//==================================================================================================
//							Beckhoff Automation Poland
//									3.01.2022
//	Function block running PLC CAM procedure using hardware limit switch
//	Library: Tc3_MC2_AdvancedHoming, Tc2_MC2, 
//
//  v1.0	|| TC v 3.1.4024.22		|| First edition 
//==================================================================================================
FUNCTION_BLOCK FB_HomingLimitSwitch
VAR_IN_OUT
	Axis 										: Tc2_MC2.AXIS_REF;
END_VAR
VAR_INPUT
	bExecute									: BOOL;
	eDirection									: Tc3_MC2_AdvancedHoming.MC_Home_Direction;
	eLimitSwitchMode							: Tc3_MC2_AdvancedHoming.MC_Switch_Mode;
	eLimitSwitchSignal							: Tc3_MC2_AdvancedHoming.MC_Ref_Signal_Ref;
	lrVelocity									: LREAL;
	lrSetPosition								: LREAL;
	tTimeLimit									: TIME;
	lrDistanceLimit								: LREAL;
	lrTorqueLimit								: LREAL;
	lrDistance									: LREAL;
END_VAR                             		
VAR_OUTPUT                              		
	bDone										: BOOL;
	bBusy										: BOOL;
	bCommandAborted								: BOOL;
	bError										: BOOL;
	nErrorID									: UDINT;
END_VAR
VAR
//=========================== Common ============================
	nStep										: UDINT;
	stParameter									: Tc3_MC2_AdvancedHoming.MC_HomingParameter;
	stOptions									: Tc3_MC2_AdvancedHoming.ST_Home_Options4;
	mcStepLimitSwitch							: Tc3_MC2_AdvancedHoming.MC_StepLimitSwitch;
//=========================== Finish ============================
	mcFinishHoming								: Tc3_MC2_AdvancedHoming.MC_FinishHoming;
//============================ Abort ============================
	mcAbortHoming								: Tc3_MC2_AdvancedHoming.MC_AbortHoming;
//========================== Internal ===========================
    {attribute 'hide'}
	nErrorID_Int								: UDINT;
//===============================================================
END_VAR

//====== Call FBs outside CASE - easier debugging ===============
mcStepLimitSwitch(	Axis						:= Axis, 
					Parameter					:= stParameter,
					LimitSwitchMode				:= eLimitSwitchMode, 
					LimitSwitchSignal			:= eLimitSwitchSignal);
                                        		
mcFinishHoming(	Axis							:= Axis, 
				Parameter						:= stParameter);
				                        	
mcAbortHoming(	Axis							:= Axis, 
				Parameter						:= stParameter);
				
//============== CASE instruction - step machine ================
CASE nStep OF
	
	0: // Wait for command
	
		IF bExecute THEN
			bBusy								:= TRUE;
				
			mcStepLimitSwitch(	Axis			:= Axis, 
								Parameter		:= stParameter,
								Execute			:= TRUE,
								Direction		:= eDirection,  
								Velocity		:= lrVelocity,
								SetPosition		:= lrSetPosition, 
								TimeLimit		:= tTimeLimit, 
								DistanceLimit	:= lrDistanceLimit,
								TorqueLimit		:= lrTorqueLimit,  
								Options			:= stOptions);
								
			// Latch finish parameters
			mcFinishHoming.Distance				:= lrDistance;
			mcFinishHoming.Velocity				:= lrVelocity;
						
			nStep								:= 1000;

		END_IF
	
	1000: // Wait till end
	
		IF mcStepLimitSwitch.Done THEN
			mcStepLimitSwitch.Execute			:= FALSE;
			nStep 								:= 3000;
		END_IF
		
		IF mcStepLimitSwitch.CommandAborted THEN
			mcStepLimitSwitch.Execute			:= FALSE;
			bBusy 								:= FALSE;
			bCommandAborted						:= TRUE;
			nStep 								:= 6000;
		END_IF
		
		IF mcStepLimitSwitch.Error THEN
			mcStepLimitSwitch.Execute			:= FALSE;
			nErrorID_Int						:= mcStepLimitSwitch.ErrorID;
			nStep 								:= 4000;
		END_IF
		
	3000: // MC_FinishHoming
	
		mcFinishHoming.Execute					:= TRUE;				
		nStep									:= nStep + 10;
		
	3010: // Wait till end
	
		IF mcFinishHoming.Done THEN
			mcFinishHoming.Execute				:= FALSE;
			bBusy 								:= FALSE;
			bDone 								:= TRUE;
			nStep 								:= 5000;
		END_IF
		
		IF mcFinishHoming.CommandAborted THEN
			mcFinishHoming.Execute				:= FALSE;
			bBusy 								:= FALSE;
			bCommandAborted						:= TRUE;
			nStep 								:= 6000;
		END_IF
		
		IF mcFinishHoming.Error THEN
			mcFinishHoming.Execute				:= FALSE;
			bBusy 								:= FALSE;
			bError								:= TRUE;
			nErrorID							:= mcFinishHoming.ErrorID;
			nStep 								:= 10000;
		END_IF	
		
	4000: // MC_AbortHoming
	
		mcAbortHoming.Execute					:= TRUE;				
		nStep									:= nStep + 10;
		
	4010: // Wait till end
	
		// No matter what is the end, we go to error State
		IF NOT mcAbortHoming.Busy THEN
			mcAbortHoming.Execute				:= FALSE;
			bBusy 								:= FALSE;
			bError								:= TRUE;
			nErrorID							:= nErrorID_Int;			
			nStep								:= 10000;
		END_IF
		
	5000: // Done
	
		bDone									:= bExecute;
		IF NOT bExecute THEN
			nStep 								:= 0;
		END_IF	
	
	6000: // Command Aborted
	
		bCommandAborted							:= bExecute;
		IF NOT bExecute THEN
			nStep 								:= 0;
		END_IF
		
	10000..20000: // Error
	
		bError									:= bExecute;
		IF NOT bExecute THEN
			nErrorID							:= 0;
			nErrorID_Int						:= 0;
			nStep 								:= 0;
		END_IF
		
END_CASE
//===============================================================

END_FUNCTION_BLOCK

(* stored: Version 1.2.0.0, ProductVersion 3.1.4026.13, FileIdentifier 8404afb12473157dedd338e275aa6d3a09d71205, FileSignature 084f28f206acc7f3e59dcc752f000e573b742996fc81463785b490fd47eb8845b401fc7b1bc651d1fb2f95f946f6ca4555927b76003c0df2a443e65d95f0083c1004aed9b24d5cbaf56c0a25a0704d30c3531803e225ca04cc5052aac3d804606e345924a0f536247bf48b33e71ce57d48b377f22bb651c923bf6f614390b1e17bf8da0bfa73126120a3dadc10d13807ab4a97991c2c8cf931a1544e712d12b7147079d33b8ca1c3d087b5199fcb1cbe96fec994bbda44e2cc128b670dab42e5df9f70a4a93e0cb3a3aee05ffe30c477620879b923ef864b283530cee6c182d3272e70f7bca6964e5b8ae8327d3904d25d39984ece7579725b870bfaaab9ea79
   POU FB_HomingLimitSwitch: Id {550df31e-dddc-4572-854f-219923240461}, SpecialFunc None *)
